{attribute 'GeneratedUsingTerminal: EPP1321-0060-0016'}
{attribute addProperty BoxType "EPP1321-0060-0016"}
{attribute addProperty Id "EtcSlaveTerminalBaseInfoDataAT %I*InfoData_6F19DB2B2"}
{attribute addProperty CRC "2874840167"}
{attribute addProperty Size "2"}
TYPE EPP1321_AB5A9467 EXTENDS EtcSlaveTerminalBase :
STRUCT
	{attribute addProperty Name "InfoData"}
	InfoData : InfoData_6F19DB2B;
END_STRUCT
END_TYPE

(* stored: Version 1.2.0.0, ProductVersion 3.1.4024.9
   DUT EPP1321_AB5A9467: Id {d84a4943-e6d6-4979-a22e-9b8dd2c2bf7f} *)
